Universal Robots PolyScope program: punto3.urp

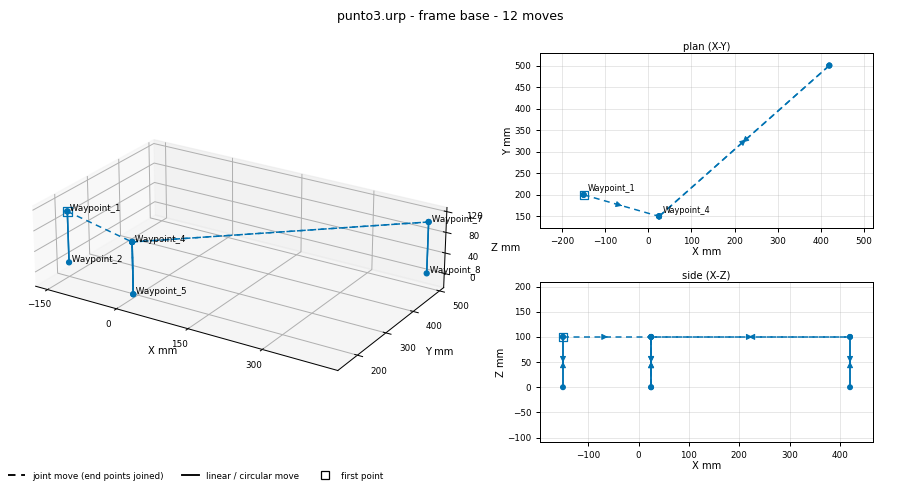
[picture p0: tool path of punto3.urp in frame base, 12 of 12 moves have a stored position in this frame; points joined in program order, loops and branches not executed]
Program punto3 (installation=default directory=/ursim/programs createdIn=3.15.8.106339 lastSavedIn=3.15.8.106339 robotSerialNumber=2018359999)
Calibrated DH parameters: a=[0, -0.425, -0.39225, 0, 0, 0]; d=[0.089159, 0, 0, 0.10915, 0.09465, 0.0823]; alpha=[1.570796, 0, 0, 1.570796, -1.570796, 0]; deltaTheta=[0, 0, 0, 0, 0, 0]
Robot Program (runOnlyOnce=false)
  Loop Forever
    MoveJ speed 60 deg/s, acceleration 80 deg/s^2 (useActiveTCP=true)
      Waypoint Waypoint_1: TCP in base x=-150 y=200 z=100 mm, rx=0 ry=-3.14 rz=0 rad; joints [-79.11, -93.879, -238.665, 62.526, 89.91, 10.89] deg; flange x=-149.761 y=200 z=250 mm, rx=0 ry=-3.14 rz=0 rad
    MoveL speed 250 mm/s, acceleration 1200 mm/s^2 (useActiveTCP=true) feature=Base
      Waypoint Waypoint_2: TCP in base x=-150 y=200 z=0 mm, rx=0 ry=-3.14 rz=0 rad; joints [-79.11, -84.038, -230.512, 44.533, 89.91, 10.89] deg; flange x=-149.761 y=200 z=150 mm, rx=0 ry=-3.14 rz=0 rad
      Set DigitalOutput pin=digital_out[0]; digitalValue=1
      Waypoint Waypoint_3: TCP in base x=-150 y=200 z=100 mm, rx=0 ry=-3.14 rz=0 rad; joints [-79.11, -93.879, -238.665, 62.526, 89.91, 10.89] deg; flange x=-149.761 y=200 z=250 mm, rx=0 ry=-3.14 rz=0 rad
    MoveJ speed 60 deg/s, acceleration 80 deg/s^2 (useActiveTCP=true)
      Waypoint Waypoint_4: TCP in base x=25 y=150 z=100 mm, rx=0 ry=-3.14 rz=0 rad; joints [-145.446, -112.382, -225.141, 67.597, 89.948, -55.446] deg; flange x=25.239 y=150 z=250 mm, rx=0 ry=-3.14 rz=0 rad
    MoveL speed 250 mm/s, acceleration 1200 mm/s^2 (useActiveTCP=true) feature=Base
      Waypoint Waypoint_5: TCP in base x=25 y=150 z=0 mm, rx=0 ry=-3.14 rz=0 rad; joints [-145.446, -100.797, -214.8, 45.672, 89.948, -55.446] deg; flange x=25.239 y=150 z=150 mm, rx=0 ry=-3.14 rz=0 rad
      Set DigitalOutput pin=digital_out[0]; digitalValue=0
      Waypoint Waypoint_6: TCP in base x=25 y=150 z=100 mm, rx=0 ry=-3.14 rz=0 rad; joints [-145.446, -112.382, -225.141, 67.597, 89.948, -55.446] deg; flange x=25.239 y=150 z=250 mm, rx=0 ry=-3.14 rz=0 rad
    MoveJ speed 60 deg/s, acceleration 80 deg/s^2 (useActiveTCP=true)
      Waypoint Waypoint_7: TCP in base x=420 y=500 z=100 mm, rx=0 ry=-3.14 rz=0 rad; joints [-139.674, -35.393, -324.151, 89.613, 89.941, -49.674] deg; flange x=420.239 y=500 z=250 mm, rx=0 ry=-3.14 rz=0 rad
    MoveL speed 250 mm/s, acceleration 1200 mm/s^2 (useActiveTCP=true) feature=Base
      Waypoint Waypoint_8: TCP in base x=420 y=500 z=0 mm, rx=0 ry=-3.14 rz=0 rad; joints [-139.674, -32.979, -314.009, 77.058, 89.941, -49.674] deg; flange x=420.239 y=500 z=150 mm, rx=0 ry=-3.14 rz=0 rad
      Set DigitalOutput pin=digital_out[0]; digitalValue=1
      Waypoint Waypoint_9: TCP in base x=420 y=500 z=100 mm, rx=0 ry=-3.14 rz=0 rad; joints [-139.674, -35.393, -324.15, 89.613, 89.941, -49.674] deg; flange x=420.239 y=500 z=250 mm, rx=0 ry=-3.14 rz=0 rad
    MoveJ speed 60 deg/s, acceleration 80 deg/s^2 (useActiveTCP=true)
      Waypoint Waypoint_4: TCP in base x=25 y=150 z=100 mm, rx=0 ry=-3.14 rz=0 rad; joints [-145.446, -112.382, -225.141, 67.597, 89.948, -55.446] deg; flange x=25.239 y=150 z=250 mm, rx=0 ry=-3.14 rz=0 rad
      MoveJ speed 60 deg/s, acceleration 80 deg/s^2 (useActiveTCP=true)
        Waypoint Waypoint_5: TCP in base x=25 y=150 z=0 mm, rx=0 ry=-3.14 rz=0 rad; joints [-145.446, -100.797, -214.8, 45.672, 89.948, -55.446] deg; flange x=25.239 y=150 z=150 mm, rx=0 ry=-3.14 rz=0 rad
        Set DigitalOutput pin=digital_out[0]; digitalValue=0
        Waypoint Waypoint_6: TCP in base x=25 y=150 z=100 mm, rx=0 ry=-3.14 rz=0 rad; joints [-145.446, -112.382, -225.141, 67.597, 89.948, -55.446] deg; flange x=25.239 y=150 z=250 mm, rx=0 ry=-3.14 rz=0 rad
    Wait DigitalInput pin=digital_in[1]; digitalValue=1
